TYPE ST_EventData1 :
STRUCT
	axis: UDINT;
	pos: LREAL;
END_STRUCT
END_TYPE

(* stored: Version 1.1.0.1, ProductVersion 3.1.0.12
   DUT ST_EventData1: Id {53f9c1e4-6898-46dc-ba94-3314b23a1fde} *)
